(* PLC project Evolved Test, Almighty ZRT11 TEST PLC Program 0.1.23.456 *)
(* stored: creationDateTime 1990-01-01T12:00:00, modificationDateTime 2016-04-10T17:37:00 *)

CONFIGURATION MotorExample_Motor
END_CONFIGURATION
